FUNCTION_BLOCK FB_ContainerWeu EXTENDS FB_ContainerBase
VAR_INPUT
END_VAR
VAR_OUTPUT
END_VAR
VAR
END_VAR

END_FUNCTION_BLOCK

(* stored: Version 1.1.0.1, ProductVersion 3.1.4024.3
   POU FB_ContainerWeu: Id {fb31222f-8037-4cb6-ae7a-cdb9b6d6ec9b}, SpecialFunc None *)
